(* IEC 61131-3 sources: CodesysTest/alpha/export/FBs/Components/Motors/Applied Motion/FB_AppliedMotionBagDeliveryMotor.pou, 8 files *)

(* ---- FB_AppliedMotionBagDeliveryMotor.pou.st ---- *)
(*#-#-#-#-#-#-#-#-#-#---Declaration---#-#-#-#-#-#-#-#-#-#-#-#-#*)

FUNCTION_BLOCK FB_AppliedMotionBagDeliveryMotor EXTENDS FB_AppliedMotionStepServoEIPBase
VAR_INPUT
	ack : BOOL;
	placement : BAG_DELIVERY_MOTOR_PLACEMENT;
	interconnect : BAG_DELIVERY_IC;
END_VAR
VAR_OUTPUT
	ackRequest : BOOL;
	tensionFault : BOOL;
END_VAR
VAR
	_moveDistance : BOOL;
	_moveFinal : BOOL;
	_moveDone : BOOL;
	_finalMove : BOOL;
	_bagDeliveryReset : BOOL;
	_delayTimer : TON := (PT := T#10MS);
	_state : BAG_DELIVERY_MOVE_STATES;
	_torqueMode : BOOL;
	_tensionFaultDwellTimer : TON := (PT := T#250MS);
	_tensionFaultEnabled : BOOL;
END_VAR
VAR CONSTANT
	O2_L : INT := 16#4CB2;
	O2_H : INT := 16#48B2;
	SCL_SO : INT := 16#534F;
	TORQUE_MODE_PARAM_ID : INT := 2;
	POINT2POINT_MODE_PARAM_ID : INT := 3;
	VELOCITY_THRESHOLD_FOR_TENSION_FAULT : INT := 500;
END_VAR
(*#-#-#-#-#-#-#-#-#-#---Implementation---#-#-#-#-#-#-#-#-#-#-#-#-#*)

(* ---- DisableTensionFault.m.st ---- *)
(*#-#-#-#-#-#-#-#-#-#---Declaration---#-#-#-#-#-#-#-#-#-#-#-#-#*)

METHOD DisableTensionFault
VAR_INPUT
END_VAR
(*#-#-#-#-#-#-#-#-#-#---Implementation---#-#-#-#-#-#-#-#-#-#-#-#-#*)

_tensionFaultEnabled := FALSE;

(* ---- EnableTensionFault.m.st ---- *)
(*#-#-#-#-#-#-#-#-#-#---Declaration---#-#-#-#-#-#-#-#-#-#-#-#-#*)

METHOD EnableTensionFault
VAR_INPUT
END_VAR
(*#-#-#-#-#-#-#-#-#-#---Implementation---#-#-#-#-#-#-#-#-#-#-#-#-#*)

_tensionFaultEnabled := TRUE;

(* ---- Execute.m.st ---- *)
(*#-#-#-#-#-#-#-#-#-#---Declaration---#-#-#-#-#-#-#-#-#-#-#-#-#*)

METHOD Execute
VAR_INPUT
END_VAR

(*#-#-#-#-#-#-#-#-#-#---Implementation---#-#-#-#-#-#-#-#-#-#-#-#-#*)

//
SUPER^.Execute();

// Used in state engine to delay between moves
_delayTimer();

// If motor velocity is greater then threshold for 2 seconds, fault
_tensionFaultDwellTimer(IN := _torqueMode AND (ABS(velocity) > VELOCITY_THRESHOLD_FOR_TENSION_FAULT));
IF (_tensionFaultDwellTimer.Q AND NOT HMIData.enableDryCycle) AND _tensionFaultEnabled THEN
	tensionFault := TRUE;
END_IF

// Clear Params
IF _bagDeliveryReset THEN
	_bagDeliveryReset := FALSE;
	_state := BAG_DELIVERY_MOVE_STATES.Idle;
	_delayTimer.IN := FALSE;
	commandSuccessful := FALSE;
	tensionFault := FALSE;
	ackRequest := FALSE;
	ack := FALSE;
END_IF

//
CASE _state OF
	BAG_DELIVERY_MOVE_STATES.Idle:
		IF _moveDistance THEN
			_moveDistance := FALSE;
			_state := BAG_DELIVERY_MOVE_STATES.SetToPointToPointMode;
			commandSuccessful := FALSE;
		END_IF

	BAG_DELIVERY_MOVE_STATES.SetToPointToPointMode:
		IF EIP THEN
			IF RearMotor THEN
				TriggerPointToPointMode();
			END_IF
			IF commandSuccessful OR NOT RearMotor THEN
				commandSuccessful := FALSE;
				_state := BAG_DELIVERY_MOVE_STATES.AckPointToPointMode;
			END_IF
		ELSIF NOT EIP THEN
			TriggerPointToPointMode();
			IF commandSuccessful THEN
				commandSuccessful := FALSE;
				_state := BAG_DELIVERY_MOVE_STATES.WaitAfterSettingOutputOff;
			END_IF
		END_IF

	BAG_DELIVERY_MOVE_STATES.WaitAfterSettingOutputOff:
		IF commandSuccessful THEN
			_state := BAG_DELIVERY_MOVE_STATES.MoveMotor;
		END_IF

	BAG_DELIVERY_MOVE_STATES.AckPointToPointMode:
		_delayTimer.PT := T#10MS;
		_delayTimer.IN := TRUE;
		IF _delayTimer.Q THEN
			ackRequest := TRUE; // Request acknowledgment from parent class
			IF ack THEN // Parent class acknowledges this motor and sibling are ready to move
				ackRequest := FALSE;
				_delayTimer.IN := FALSE;
				_state := BAG_DELIVERY_MOVE_STATES.MoveMotor;
			END_IF
		END_IF

	BAG_DELIVERY_MOVE_STATES.MoveMotor:
		FeedToLength();
		_state := BAG_DELIVERY_MOVE_STATES.WaitAfterMovingMotor;

	BAG_DELIVERY_MOVE_STATES.WaitAfterMovingMotor:
		IF NOT _moveFinal THEN
			IF commandSuccessful THEN
				commandSuccessful := FALSE;
				_moveDone := TRUE;
				_state := BAG_DELIVERY_MOVE_STATES.Idle;
			END_IF
		ELSE
			IF commandSuccessful AND InPosition THEN
				_delayTimer.PT := T#10MS;
				_delayTimer.IN := TRUE;
				IF _delayTimer.Q THEN
					_delayTimer.IN := FALSE;
					commandSuccessful := FALSE;
					_state := BAG_DELIVERY_MOVE_STATES.SetToTorqueMode;
				END_IF
			END_IF
		END_IF

	BAG_DELIVERY_MOVE_STATES.SetToTorqueMode:
		IF EIP THEN
			IF RearMotor THEN
				TriggerTorqueMode();
			END_IF
			IF commandSuccessful OR NOT RearMotor THEN
				commandSuccessful := FALSE;
				_state := BAG_DELIVERY_MOVE_STATES.WaitAfterSettingOutputOn;
			END_IF
		ELSE
			TriggerTorqueMode();
			IF commandSuccessful THEN
				commandSuccessful := FALSE;
				_state := BAG_DELIVERY_MOVE_STATES.WaitAfterSettingOutputOn;
			END_IF
		END_IF

	BAG_DELIVERY_MOVE_STATES.WaitAfterSettingOutputOn:
		IF EIP THEN
			_delayTimer.PT := T#10MS;
			_delayTimer.IN := TRUE;
			IF _delayTimer.Q THEN
				_moveDone := TRUE;
				_moveFinal := FALSE;
				_delayTimer.IN := FALSE;
				_state := BAG_DELIVERY_MOVE_STATES.Idle;
			END_IF
		ELSE
			_moveDone := TRUE;
			_state := BAG_DELIVERY_MOVE_STATES.Idle;
		END_IF
END_CASE

(* ---- MoveDistanceFinal.m.st ---- *)
(*#-#-#-#-#-#-#-#-#-#---Declaration---#-#-#-#-#-#-#-#-#-#-#-#-#*)

METHOD MoveDistanceFinal
VAR_INPUT
    distance : REAL;        //Distance to move in inches
    acceleration : INT;        //Acceleration in RPM/sec
    deceleration : INT;        //Deceleration in RPM/sec
    velocity : INT;            //Velocity in .25RPM
END_VAR
(*#-#-#-#-#-#-#-#-#-#---Implementation---#-#-#-#-#-#-#-#-#-#-#-#-#*)

// Return if a rear motor using cable or a command is running
IF RearMotor AND NOT EIP THEN
	RETURN;
END_IF

//
_moveDone := FALSE;
_moveFinal := TRUE;
_moveDistance := TRUE;
_state := BAG_DELIVERY_MOVE_STATES.Idle;

//
distanceToMoveInSteps := REAL_TO_DINT((distance) * stepsPerInchSetpoint);
IF reversePolarity THEN
    distanceToMoveInSteps := distanceToMoveInSteps * -1;
END_IF

//
commandSuccessful := FALSE;
pointToPointAccelSetpoint := acceleration;
pointToPointDecelSetpoint := deceleration;
currentLimit := defaultCurrentSetpoint;
velocitySetpoint := velocity;

(* ---- Reset.m.st ---- *)
(*#-#-#-#-#-#-#-#-#-#---Declaration---#-#-#-#-#-#-#-#-#-#-#-#-#*)

METHOD Reset : BOOL
VAR_INPUT
END_VAR
(*#-#-#-#-#-#-#-#-#-#---Implementation---#-#-#-#-#-#-#-#-#-#-#-#-#*)

_restoreToDefault := TRUE;

(* ---- TriggerPointToPointMode.m.st ---- *)
(*#-#-#-#-#-#-#-#-#-#---Declaration---#-#-#-#-#-#-#-#-#-#-#-#-#*)

METHOD TriggerPointToPointMode
VAR_INPUT
END_VAR

(*#-#-#-#-#-#-#-#-#-#---Implementation---#-#-#-#-#-#-#-#-#-#-#-#-#*)

IF EIP THEN
	parameter1 := POINT2POINT_MODE_PARAM_ID;
	commands.SendQAndExecute := TRUE;
ELSE
	sclCommand := SCL_SO;
	parameter1 := O2_H;
	commands.SendHostCommand := TRUE;
END_IF

(* ---- TriggerTorqueMode.m.st ---- *)
(*#-#-#-#-#-#-#-#-#-#---Declaration---#-#-#-#-#-#-#-#-#-#-#-#-#*)

METHOD TriggerTorqueMode
VAR_INPUT
END_VAR
(*#-#-#-#-#-#-#-#-#-#---Implementation---#-#-#-#-#-#-#-#-#-#-#-#-#*)

IF EIP THEN
	sclCommand := 0;
	parameter1 := TORQUE_MODE_PARAM_ID;
	commands.SendQAndExecute := TRUE;
ELSE
	sclCommand := SCL_SO;
	parameter1 := O2_L;
	commands.SendHostCommand := TRUE;
END_IF
